	FUNCTION_BLOCK FB 335
	TITLE =G235M INLET SLIDE GERM 7
	//COPYRIGHT:    (C) 2009  BUHLER AG, CH-9240 UZWIL, SWITZERLAND
	//
	//PRODUCT:      WinCoS_BIW01_09
	//
	//TITLE:        INLET SLIDE GERM 7
	//                Machine group control
	//                Maschinengruppensteuerung
	//
	//--------------------------------------------------------------------------------
	//
	//IDENT:        AUTHOR:             DEPT:                              DATE:
	//
	//P01_FB335.1.0 K.Renz              CSB41                              13.Jan.2010
	//             1st Release
	//
	//--------------------------------------------------------------------------------
	//
	//PURPOSE:
	//
	//MANUAL :
	//
	//RESTRICTIONS:
	//
	//--------------------------------------------------------------------------------
	AUTHOR  : KR
	FAMILY  : USW
	VERSION : 9.9


	VAR
	  Gr       : FB10;	//Standard interface to group
	  InOutValue1    : DINT; //Data for user
	  InOutValue2    : DINT; //Data for user
	  OutWayConflict : BOOL;	//Data for user
	  OutSelectionOk : BOOL;	//Data for user
	  CmdNewValue : BOOL;	//Data for user
	  CmdNewJob   : BOOL;	//Data for user
	  OutCodeOK   : BOOL;	//Data for user
	  InEndOfJob  : BOOL ;	//Data for user
	  staWayOk      : BOOL ;	//Data for user
	  EdgeStartRelease : BOOL ;	//Data for user
	  USW8  : BOOL;	//Data for user
	  USW9 : BOOL;	//Data for user
	  USW10: BOOL;	//Data for user
	  USW11: BOOL;	//Data for user
	  USW12: BOOL;	//Data for user
	  USW13: BOOL;	//Data for user
	  USW14: BOOL;	//Data for user
	  USW15: BOOL;	//Data for user
	     #A_2702_BZS13 : FB14;   // DigInpCont
	     #A_2702_BZS14 : FB14;   // DigInpCont
	     #A_2702_BZS15 : FB14;   // DigInpCont
	     #A_2702_MXZ01 : FB12;   // Motor
	     #A_2702_QYS21 : FB14;   // DigInpCont
	     #A_2702_QYS22 : FB14;   // DigInpCont
	END_VAR
	VAR_TEMP
	   tmpEnable		: BOOL;
	   tmpFlag  		: BOOL;
	   tmpCmdNext		: BOOL;
	   tmpLocal  		: BOOL;
	   tmpAspOk  		: BOOL;
	   tmpHWStop 		: BOOL;
	   tmpInstanzDBNo       : INT ;
	END_VAR
	BEGIN
	NETWORK
	TITLE =
	NETWORK
	TITLE =Read command from group control
	//Parameter
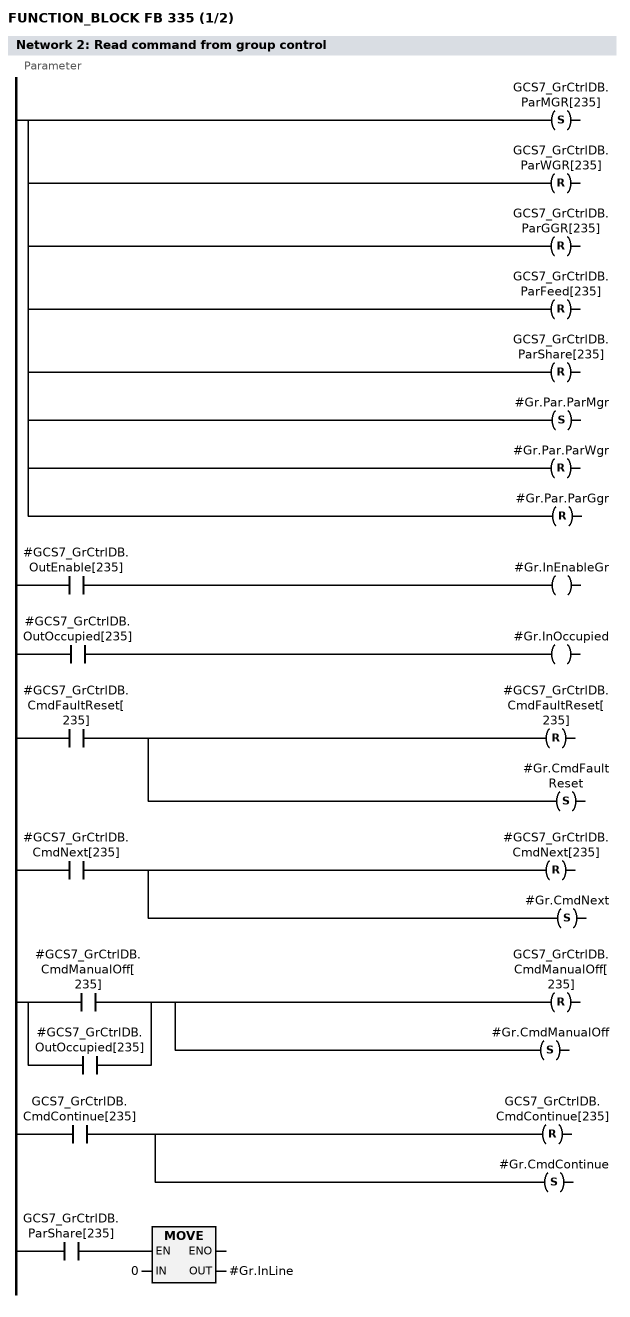
	      SET;
	      S   GCS7_GrCtrlDB.ParMGR[235];
	      R   GCS7_GrCtrlDB.ParWGR[235];
	      R   GCS7_GrCtrlDB.ParGGR[235];
	      R   GCS7_GrCtrlDB.ParFeed[235];
	      R   GCS7_GrCtrlDB.ParShare[235];
	      S   #Gr.Par.ParMgr;
	      R   #Gr.Par.ParWgr;
	      R   #Gr.Par.ParGgr;
	//Command
	      U   #GCS7_GrCtrlDB.OutEnable[235];
	      =   #Gr.InEnableGr;
	      U   #GCS7_GrCtrlDB.OutOccupied[235];
	      =   #Gr.InOccupied;
	      U   #GCS7_GrCtrlDB.CmdFaultReset[235];
	      R   #GCS7_GrCtrlDB.CmdFaultReset[235];
	      S   #Gr.CmdFaultReset;
	      U  #GCS7_GrCtrlDB.CmdNext[235];
	      R   #GCS7_GrCtrlDB.CmdNext[235];
	      S   #Gr.CmdNext;
	      U   #GCS7_GrCtrlDB.CmdManualOff[235];
	      O   #GCS7_GrCtrlDB.OutOccupied[235];
	      R   GCS7_GrCtrlDB.CmdManualOff[235];
	      S   #Gr.CmdManualOff;
	      U  GCS7_GrCtrlDB.CmdContinue[235];
	      R   GCS7_GrCtrlDB.CmdContinue[235];
	      S   #Gr.CmdContinue;
	//Init Line Number
	      U   GCS7_GrCtrlDB.ParShare[235];
	      SPBN WE00;
	      L     0;
	      T     #Gr.InLine;
	WE00: NOP   0;
	NETWORK
	TITLE =Call Methode Control
	// 1. Handle Interface PCControl
	// 2. Prepare mode --> ModePassive,ModeActive,ModeIdling
	// 3. Reset global flags of the group
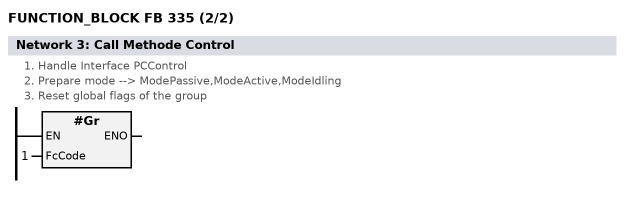
	      CALL #Gr (
	           FcCode                   := 1);
	NETWORK
	TITLE =Restart Idling Time
		L  #Gr.Par.ParIdling;
		L  2;
		>=I;
		SPB IdTm;
		T  #Gr.Par.ParIdling;
	IdTm:   NOP 0;
	      CLR;
	      S    #Gr.CmdRestartIdling;
	NETWORK
	TITLE =Prepare global flags
	NETWORK
	TITLE =Set Pattern (Target position)
	NETWORK
	TITLE =Interlocking WayOk
	//
	NETWORK
	TITLE =Interlocking Autostart
		CLR;
		R   #Gr.OutAutostart;
	NETWORK
	TITLE =Interlocking Enable
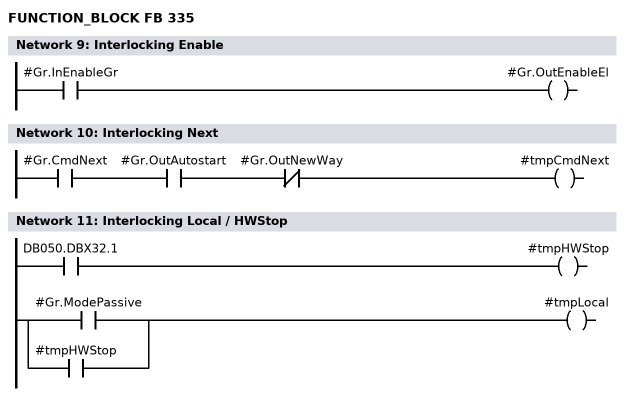
	      U     #Gr.InEnableGr;
	      =     #Gr.OutEnableEl;

	NETWORK
	TITLE =Interlocking Next
	      U     #Gr.CmdNext;
	      U     #Gr.OutAutostart;
	      UN    #Gr.OutNewWay;
	      =    #tmpCmdNext;

	NETWORK
	TITLE =Interlocking Local / HWStop
	      U    DB050.DBX32.1;
	      =    #tmpHWStop;

	      U    #Gr.ModePassive;
	      O    #tmpHWStop;
	      =    #tmpLocal;

	NETWORK
	TITLE =Interlocking Start Warning
	      NOP 0;
	//- Restart after fault --
	      U     #Gr.CmdFaultReset;
	      U     #Gr.VarFault;
	      S       "SYS_StartWarningDB".Area[8].CmdResetStartWarning;
	//- Run Timer --
	      AUF "G235M";
	      CALL  FB100 , DB100(
	       InModeHigher :=FALSE,
	       InArea     :=8,
	       InEnable   :=#Gr.OutEnableEl,
	       InLocal    :=#tmpLocal,
	       InStarted  :=#Gr.VarStarted,
	       InCmdNext  :=#tmpCmdNext,
	       OutCmdNext :=#tmpCmdNext,
	       OutStartwarning:=#Gr.VarStartWarning);
	//- Store Startwarning done  --
	//- Reset Autostart --
	      U     "SYS_StartWarningDB".TmpArea.OutStartReleaseRunningL;
	      FN    #EdgeStartRelease;
	      U     #Gr.VarFault;
	      R     #Gr.OutAutostart;
	NETWORK
	TITLE ==A-2702-BZS13 : DISCHARGE CHUTE PARKING POSITION
	NOP 0;
	//-InLocal---
	      U     #tmpLocal;
	      =     #A_2702_BZS13.InLocal;
	//
	//-Monitoring---
	      CLR;
	      =      #A_2702_BZS13.InMonTrue;
	      CLR;
	      =      #A_2702_BZS13.InMonFalse;
	//
	//-PreAlarm---
	      CLR;
	      =      #A_2702_BZS13.InPreAlarmTrue;
	      CLR;
	      =      #A_2702_BZS13.InPreAlarmFalse;
	//
	//-Additional commands---
	//      CLR
	//      S     #A_2702_BZS13.CmdRunTimeOutTime
	//
	//-Read inputs---
	      U     E 718.2;
	      =     #A_2702_BZS13.InpTrue;
	       U     PLC_DPInfo.Master[1].SlavesError[73];
	       =       #A_2702_BZS13.InDPFault;
	//
	//-Set Parameters---
	//
	//-Call object control---
	      CALL  #A_2702_BZS13;
	//
	//-Write outputs---
	NETWORK
	TITLE ==A-2702-BZS14 : DISCHARGE CHUTE LEFT SIDE
	NOP 0;
	//-InLocal---
	      U     #tmpLocal;
	      =     #A_2702_BZS14.InLocal;
	//
	//-Monitoring---
	      CLR;
	      =      #A_2702_BZS14.InMonTrue;
	      CLR;
	      =      #A_2702_BZS14.InMonFalse;
	//
	//-PreAlarm---
	      CLR;
	      =      #A_2702_BZS14.InPreAlarmTrue;
	      CLR;
	      =      #A_2702_BZS14.InPreAlarmFalse;
	//
	//-Additional commands---
	//      CLR
	//      S     #A_2702_BZS14.CmdRunTimeOutTime
	//
	//-Read inputs---
	      U     E 718.3;
	      =     #A_2702_BZS14.InpTrue;
	       U     PLC_DPInfo.Master[1].SlavesError[73];
	       =       #A_2702_BZS14.InDPFault;
	//
	//-Set Parameters---
	//
	//-Call object control---
	      CALL  #A_2702_BZS14;
	//
	//-Write outputs---
	NETWORK
	TITLE ==A-2702-BZS15 : DISCHARGE CHUTE RIGHT SIDE
	NOP 0;
	//-InLocal---
	      U     #tmpLocal;
	      =     #A_2702_BZS15.InLocal;
	//
	//-Monitoring---
	      CLR;
	      =      #A_2702_BZS15.InMonTrue;
	      CLR;
	      =      #A_2702_BZS15.InMonFalse;
	//
	//-PreAlarm---
	      CLR;
	      =      #A_2702_BZS15.InPreAlarmTrue;
	      CLR;
	      =      #A_2702_BZS15.InPreAlarmFalse;
	//
	//-Additional commands---
	//      CLR
	//      S     #A_2702_BZS15.CmdRunTimeOutTime
	//
	//-Read inputs---
	      U     E 718.4;
	      =     #A_2702_BZS15.InpTrue;
	       U     PLC_DPInfo.Master[1].SlavesError[73];
	       =       #A_2702_BZS15.InDPFault;
	//
	//-Set Parameters---
	//
	//-Call object control---
	      CALL  #A_2702_BZS15;
	//
	//-Write outputs---
	NETWORK
	TITLE ==A-2702-MXZ01 : CHUTE DRIVE
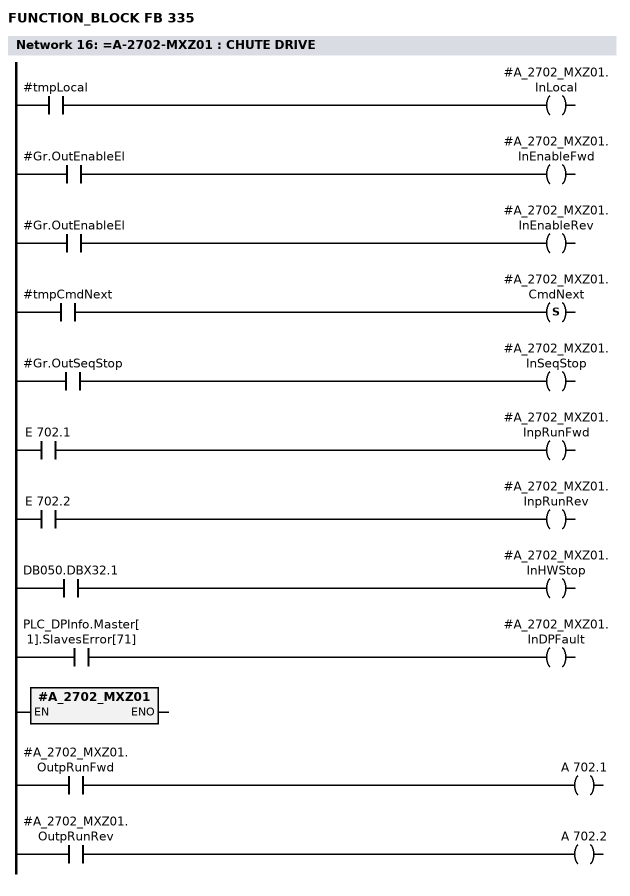
	NOP 0;
	//-InLocal---
	      U     #tmpLocal;
	      =     #A_2702_MXZ01.InLocal;
	//
	//-Interlocking---
	      U     #Gr.OutEnableEl;
	      =     #A_2702_MXZ01.InEnableFwd;
	      U     #Gr.OutEnableEl;
	      =     #A_2702_MXZ01.InEnableRev;
	//
	      U    #tmpCmdNext;
	      S     #A_2702_MXZ01.CmdNext;
	//
	      U     #Gr.OutSeqStop;
	      =     #A_2702_MXZ01.InSeqStop;
	//
	//-Read inputs---
	      U     E 702.1;
	      =     #A_2702_MXZ01.InpRunFwd;
	      U     E 702.2;
	      =     #A_2702_MXZ01.InpRunRev;
	      U   DB050.DBX32.1;
	      =     #A_2702_MXZ01.InHWStop;
	       U     PLC_DPInfo.Master[1].SlavesError[71];
	       =       #A_2702_MXZ01.InDPFault;
	//
	//-Set Parameters---
	//
	//-Call object control---
	      CALL  #A_2702_MXZ01;
	//
	//-Write outputs---
	      U     #A_2702_MXZ01.OutpRunFwd;
	      =     A 702.1;
	      U     #A_2702_MXZ01.OutpRunRev;
	      =     A 702.2;
	NETWORK
	TITLE ==A-2702-QYS21 : DISCHARGE CHUTE LEFT SIDE
	NOP 0;
	//-InLocal---
	      U     #tmpLocal;
	      =     #A_2702_QYS21.InLocal;
	//
	//-Monitoring---
	      CLR;
	      =      #A_2702_QYS21.InMonTrue;
	      CLR;
	      =      #A_2702_QYS21.InMonFalse;
	//
	//-PreAlarm---
	      CLR;
	      =      #A_2702_QYS21.InPreAlarmTrue;
	      CLR;
	      =      #A_2702_QYS21.InPreAlarmFalse;
	//
	//-Additional commands---
	//      CLR
	//      S     #A_2702_QYS21.CmdRunTimeOutTime
	//
	//-Read inputs---
	      U     E 705.5;
	      =     #A_2702_QYS21.InpTrue;
	       U     PLC_DPInfo.Master[1].SlavesError[71];
	       =       #A_2702_QYS21.InDPFault;
	//
	//-Set Parameters---
	//
	//-Call object control---
	      CALL  #A_2702_QYS21;
	//
	//-Write outputs---
	NETWORK
	TITLE ==A-2702-QYS22 : DISCHARGE CHUTE RIGHT SIDE
	NOP 0;
	//-InLocal---
	      U     #tmpLocal;
	      =     #A_2702_QYS22.InLocal;
	//
	//-Monitoring---
	      CLR;
	      =      #A_2702_QYS22.InMonTrue;
	      CLR;
	      =      #A_2702_QYS22.InMonFalse;
	//
	//-PreAlarm---
	      CLR;
	      =      #A_2702_QYS22.InPreAlarmTrue;
	      CLR;
	      =      #A_2702_QYS22.InPreAlarmFalse;
	//
	//-Additional commands---
	//      CLR
	//      S     #A_2702_QYS22.CmdRunTimeOutTime
	//
	//-Read inputs---
	      U     E 705.6;
	      =     #A_2702_QYS22.InpTrue;
	       U     PLC_DPInfo.Master[1].SlavesError[71];
	       =       #A_2702_QYS22.InDPFault;
	//
	//-Set Parameters---
	//
	//-Call object control---
	      CALL  #A_2702_QYS22;
	//
	//-Write outputs---
	NETWORK
	TITLE =Test Fault
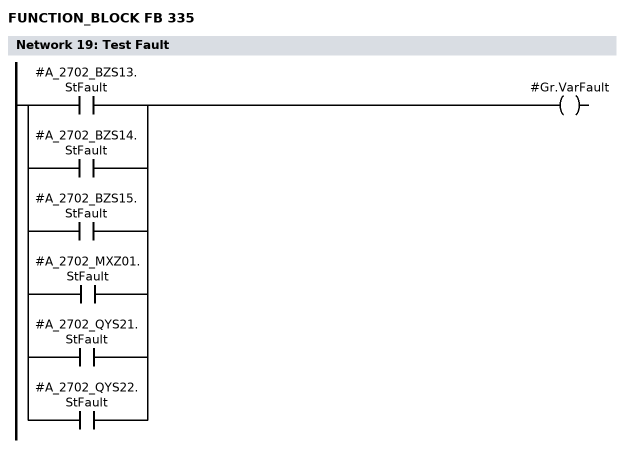
	      U     #A_2702_BZS13.StFault;
	      O     #A_2702_BZS14.StFault;
	      O     #A_2702_BZS15.StFault;
	      O     #A_2702_MXZ01.StFault;
	      O     #A_2702_QYS21.StFault;
	      O     #A_2702_QYS22.StFault;
	      =     #Gr.VarFault;
	NETWORK
	TITLE =Test Warning
	      CLR;
	      =     #Gr.OutWarning;
	NETWORK
	TITLE =Test Stopped
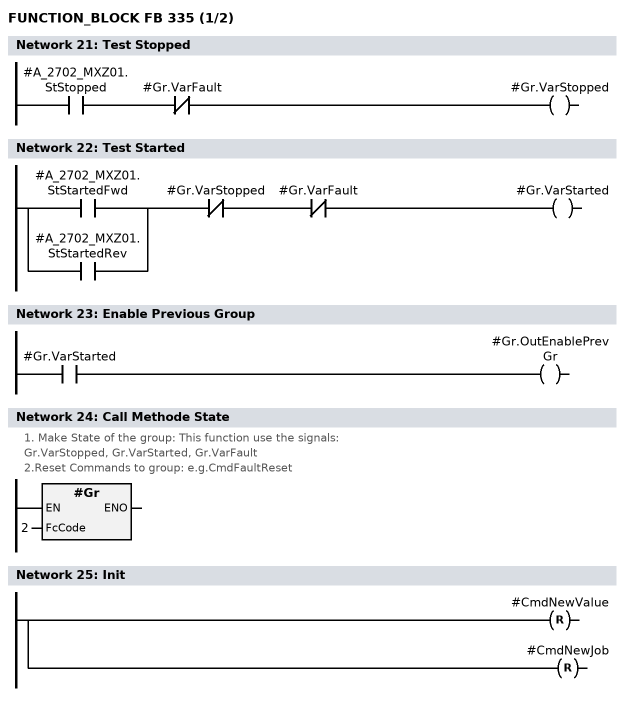
	      U     #A_2702_MXZ01.StStopped;
	      UN   #Gr.VarFault;
	      =     #Gr.VarStopped;
	NETWORK
	TITLE =Test Started
	      U(;
	      O     #A_2702_MXZ01.StStartedFwd;
	      O     #A_2702_MXZ01.StStartedRev;
	      );
	      UN  #Gr.VarStopped;
	      UN  #Gr.VarFault;
	      =     #Gr.VarStarted;
	NETWORK
	TITLE =Enable Previous Group
	      U    #Gr.VarStarted;
	      =     #Gr.OutEnablePrevGr;
	NETWORK
	TITLE =Call Methode State
	//1. Make State of the group: This function use the signals:
	//        Gr.VarStopped, Gr.VarStarted, Gr.VarFault
	//2.Reset Commands to group: e.g.CmdFaultReset
	      CALL #Gr (
	           FcCode                   := 2);
	NETWORK
	TITLE =Init
	      SET;
	      R    #CmdNewValue;
	      R    #CmdNewJob;
	NETWORK
	TITLE =Write data to group control
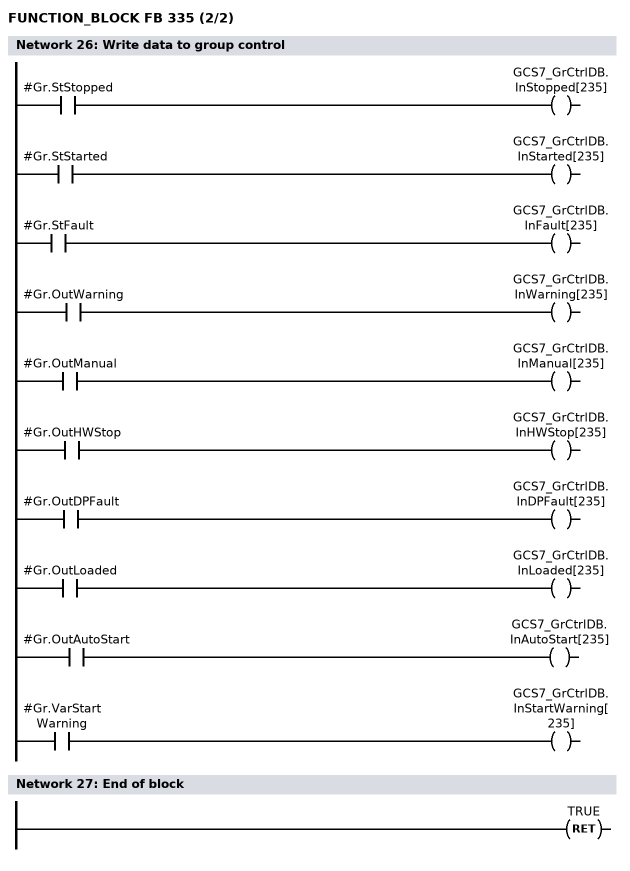
	      U   #Gr.StStopped;
	      =   GCS7_GrCtrlDB.InStopped[235];
	      U   #Gr.StStarted;
	      =   GCS7_GrCtrlDB.InStarted[235];
	      U   #Gr.StFault;
	      =   GCS7_GrCtrlDB.InFault[235];
	      U   #Gr.OutWarning;
	      =   GCS7_GrCtrlDB.InWarning[235];
	      U   #Gr.OutManual;
	      =   GCS7_GrCtrlDB.InManual[235];
	      U   #Gr.OutHWStop;
	      =   GCS7_GrCtrlDB.InHWStop[235];
	      U   #Gr.OutDPFault;
	      =   GCS7_GrCtrlDB.InDPFault[235];
	      U   #Gr.OutLoaded;
	      =   GCS7_GrCtrlDB.InLoaded[235];
	      U   #Gr.OutAutoStart;
	      =   GCS7_GrCtrlDB.InAutoStart[235];
	      U   #Gr.VarStartWarning;
	      =   GCS7_GrCtrlDB.InStartWarning[235];
	NETWORK
	TITLE =End of block

	BE

	END_FUNCTION_BLOCK
